// TIA Portal V17 export
// export: Created 2026-04-13T11:12:53.2804569Z, ExportSetting WithDefaults, DisplayName Totally Integrated Automation Portal, DisplayVersion V17 Update 4, DisplayName TIA Portal Openness, DisplayVersion V17 Update 4, DisplayName TIA Portal Version Control Interface, DisplayVersion V17, DisplayName SINAMICS Startdrive Advanced, DisplayVersion V17, DisplayName SINAMICS Startdrive G130, G150, S120, S150, SINAMICS MV, S210, DisplayVersion V17, DisplayName SINAMICS Startdrive G110M, G120, G120C, G120D, G120P, G115D, DisplayVersion V17, DisplayName STEP 7 Professional, DisplayVersion V17 Update 4, DisplayName STEP 7 Safety, DisplayVersion V17, DisplayName WinCC Professional, DisplayVersion V17 Update 4
TagTable "INCIPCS"
  INCIPCS_1设定时间 : Real  (PLC tag INCIPCS.1设定时间, HMI_连接_1, 1 s)
  INCIPCS_2设定时间 : Real  (PLC tag INCIPCS.2设定时间, HMI_连接_1, 1 s)
  INCIPCS_3设定时间 : Real  (PLC tag INCIPCS.3设定时间, HMI_连接_1, 1 s)
  INCIPCS_4设定时间 : Real  (PLC tag INCIPCS.4设定时间, HMI_连接_1, 1 s)
  INCIPCS_5设定时间 : Real  (PLC tag INCIPCS.5设定时间, HMI_连接_1, 1 s)
  INCIPCS_6设定时间 : Real  (PLC tag INCIPCS.6设定时间, HMI_连接_1, 1 s)
  INCIPCS_7设定时间 : Real  (PLC tag INCIPCS.7设定时间, HMI_连接_1, 1 s)
  INCIPCS_8设定时间 : Real  (PLC tag INCIPCS.8设定时间, HMI_连接_1, 1 s)
  INCIPCS_9设定时间 : Real  (PLC tag INCIPCS.9设定时间, HMI_连接_1, 1 s)
  INCIPCS_10设定时间 : Real  (PLC tag INCIPCS.10设定时间, HMI_连接_1, 1 s)
  INCIPCS_11设定时间 : Real  (PLC tag INCIPCS.11设定时间, HMI_连接_1, 1 s)
  INCIPCS_12设定时间 : Real  (PLC tag INCIPCS.12设定时间, HMI_连接_1, 1 s)
  INCIPCS_13设定时间 : Real  (PLC tag INCIPCS.13设定时间, HMI_连接_1, 1 s)
  INCIPCS_14设定时间 : Real  (PLC tag INCIPCS.14设定时间, HMI_连接_1, 1 s)
  INCIPCS_15设定时间 : Real  (PLC tag INCIPCS.15设定时间, HMI_连接_1, 1 s)
  INCIPCS_16设定时间 : Real  (PLC tag INCIPCS.16设定时间, HMI_连接_1, 1 s)
  INCIPCS_0计时 : Real  (PLC tag INCIPCS.0计时, HMI_连接_1, 1 s)
  INCIPCS_1计时 : Real  (PLC tag INCIPCS.1计时, HMI_连接_1, 1 s)
  INCIPCS_2计时 : Real  (PLC tag INCIPCS.2计时, HMI_连接_1, 1 s)
  INCIPCS_3计时 : Real  (PLC tag INCIPCS.3计时, HMI_连接_1, 1 s)
  INCIPCS_4计时 : Real  (PLC tag INCIPCS.4计时, HMI_连接_1, 1 s)
  INCIPCS_5计时 : Real  (PLC tag INCIPCS.5计时, HMI_连接_1, 1 s)
  INCIPCS_6计时 : Real  (PLC tag INCIPCS.6计时, HMI_连接_1, 1 s)
  INCIPCS_7计时 : Real  (PLC tag INCIPCS.7计时, HMI_连接_1, 1 s)
  INCIPCS_8计时 : Real  (PLC tag INCIPCS.8计时, HMI_连接_1, 1 s)
  INCIPCS_9计时 : Real  (PLC tag INCIPCS.9计时, HMI_连接_1, 1 s)
  INCIPCS_10计时 : Real  (PLC tag INCIPCS.10计时, HMI_连接_1, 1 s)
  INCIPCS_11计时 : Real  (PLC tag INCIPCS.11计时, HMI_连接_1, 1 s)
  INCIPCS_12计时 : Real  (PLC tag INCIPCS.12计时, HMI_连接_1, 1 s)
  INCIPCS_13计时 : Real  (PLC tag INCIPCS.13计时, HMI_连接_1, 1 s)
  INCIPCS_14计时 : Real  (PLC tag INCIPCS.14计时, HMI_连接_1, 1 s)
  INCIPCS_15计时 : Real  (PLC tag INCIPCS.15计时, HMI_连接_1, 1 s)
  INCIPCS_16计时 : Real  (PLC tag INCIPCS.16计时, HMI_连接_1, 1 s)
